// TIA Portal V17 export
// export: Created 2022-03-12T16:05:26.7716914Z, ExportSetting WithDefaults, DisplayName Totally Integrated Automation Portal, DisplayVersion V17, DisplayName TIA Portal Openness, DisplayVersion V17, DisplayName TIA Portal Version Control Interface, DisplayVersion V17, DisplayName STEP 7 Professional, DisplayVersion V17, DisplayName STEP 7 Safety, DisplayVersion V17, DisplayName WinCC Advanced / Unified PC, DisplayVersion V17
FUNCTION_BLOCK "EM00_CM01_MainOpStation"   // FB31651, LAD
TITLE = EM00_CM01_MainOpStation
{ S7_Optimized_Access := 'TRUE' }
AUTHOR : tech.team.motioncontrol@siemens.com
FAMILY : CPG
VERSION : 1.1
// Support: tech.team.motioncontrol@siemens.com
// stored: AutoNumber true, IsIECCheckEnabled false, IsRetainMemResEnabled false, MemoryReserve 100, SetENOAutomatically false, UDAEnableTagReadback false
   VAR
      instAlarm_EStop { ExternalAccessible := 'False'; ExternalVisible := 'False'; ExternalWritable := 'False'; S7_SetPoint := 'True'} : "CPG_Event";   // Alarm Event - EStop pressed (Event instance)
      instAlarm_HMI_StopPB { ExternalAccessible := 'False'; ExternalVisible := 'False'; ExternalWritable := 'False'; S7_SetPoint := 'True'} : "CPG_Event";   // Alarm Event - HMI Stop PB pressed (Event instance)
      instStatus_WaitingForStartCmd { ExternalAccessible := 'False'; ExternalVisible := 'False'; ExternalWritable := 'False'; S7_SetPoint := 'True'} : "CPG_Event";   // Status Event - waiting for start command (Event instance)
      instStatus_WaitingForResetCmd { ExternalAccessible := 'False'; ExternalVisible := 'False'; ExternalWritable := 'False'; S7_SetPoint := 'True'} : "CPG_Event";   // Status Event - waiting for reset command (Event instance)
      instAlarm_Hold_PB { ExternalAccessible := 'False'; ExternalVisible := 'False'; ExternalWritable := 'False'; S7_SetPoint := 'True'} : "CPG_Event";   // Alarm Event - HMI Held PB pressed (Event instance)
      instStatus_WaitingForUnHoldCmd { ExternalAccessible := 'False'; ExternalVisible := 'False'; ExternalWritable := 'False'; S7_SetPoint := 'True'} : "CPG_Event";   // Status Event - waiting for unhold command (Event instance)
      instTimer_StartingDelay_SC { ExternalAccessible := 'False'; ExternalVisible := 'False'; ExternalWritable := 'False'; S7_SetPoint := 'True'} : IEC_TIMER;   // IEC Timer - starting delay (demo only - used to slow state model transition)
      instTimer_CompletingDelay_SC { ExternalAccessible := 'False'; ExternalVisible := 'False'; ExternalWritable := 'False'; S7_SetPoint := 'True'} : IEC_TIMER;   // IEC Timer - completing delay (demo only - used to slow state model transition)
      instTimer_AbortingDelay_SC { ExternalAccessible := 'False'; ExternalVisible := 'False'; ExternalWritable := 'False'; S7_SetPoint := 'True'} : IEC_TIMER;   // IEC Timer - aborting delay (demo only - used to slow state model transition)
      instTimer_StoppingDelay_SC { ExternalAccessible := 'False'; ExternalVisible := 'False'; ExternalWritable := 'False'; S7_SetPoint := 'True'} : IEC_TIMER;   // IEC Timer - stopping delay (demo only - used to slow state model transition)
      instTimer_ResettingDelay_SC { ExternalAccessible := 'False'; ExternalVisible := 'False'; ExternalWritable := 'False'; S7_SetPoint := 'True'} : IEC_TIMER;   // IEC Timer - resetting delay (demo only - used to slow state model transition)
      instTimer_HoldingDelay_SC { ExternalAccessible := 'False'; ExternalVisible := 'False'; ExternalWritable := 'False'; S7_SetPoint := 'True'} : IEC_TIMER;   // IEC Timer - holding delay (demo only - used to slow state model transition)
      instTimer_UnHoldingDelay_SC { ExternalAccessible := 'False'; ExternalVisible := 'False'; ExternalWritable := 'False'; S7_SetPoint := 'True'} : IEC_TIMER;   // IEC Timer - un-holding delay (demo only - used to slow state model transition)
      instTimer_SuspendingDelay_SC { ExternalAccessible := 'False'; ExternalVisible := 'False'; ExternalWritable := 'False'; S7_SetPoint := 'True'} : IEC_TIMER;   // IEC Timer - suspending delay (demo only - used to slow state model transition)
      instTimer_UnSuspendingDelay_SC { ExternalAccessible := 'False'; ExternalVisible := 'False'; ExternalWritable := 'False'; S7_SetPoint := 'True'} : IEC_TIMER;   // IEC Timer - un-suspending delay (demo only - used to slow state model transition)
      instTimer_ClearingDelay_SC { ExternalAccessible := 'False'; ExternalVisible := 'False'; ExternalWritable := 'False'; S7_SetPoint := 'True'} : IEC_TIMER;   // IEC Timer - clearing delay (demo only - used to slow state model transition)
   END_VAR
BEGIN

REGION Network 1: *** Begin the Setpoint Management Information Section ***
END_REGION

REGION Network 2: *** Begin the Logic Section ***
END_REGION

REGION Network 3: *** Begin the Event Information Section ***
END_REGION

REGION Network 4: Alarm Event - EStop
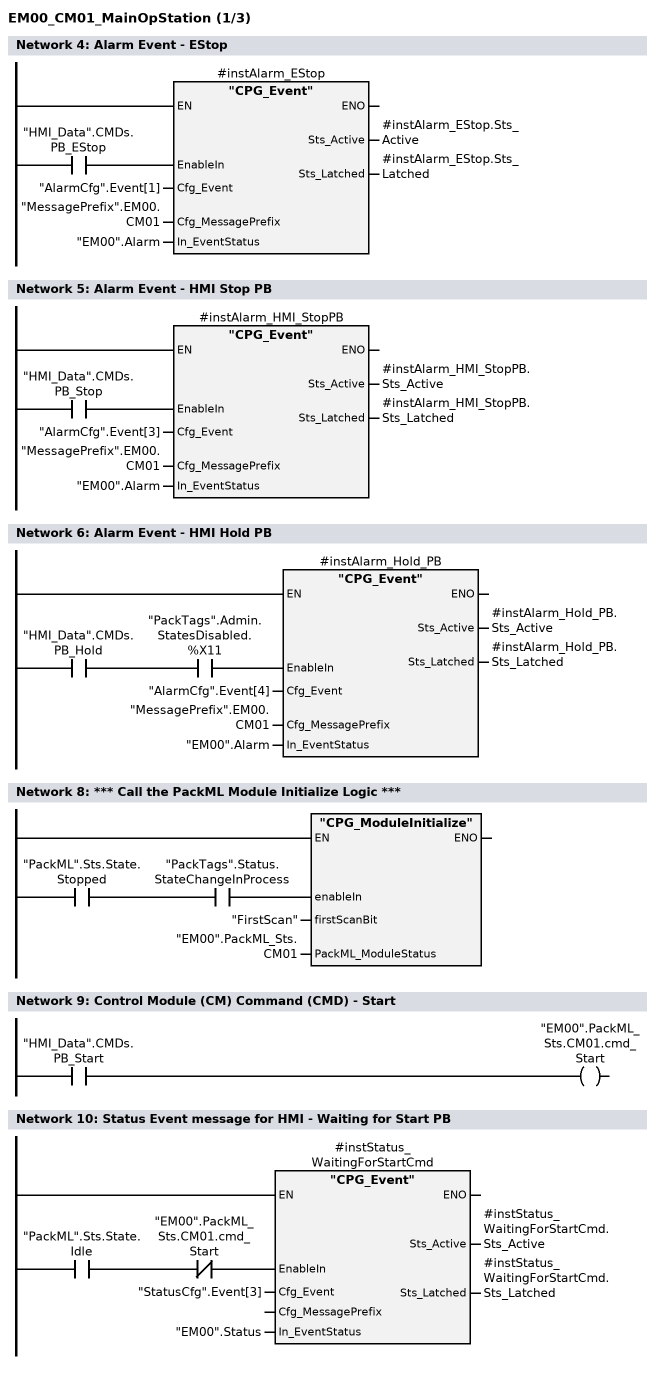
   RUNG wire#powerrail
      #instAlarm_EStop(EnableIn := wire#w1, Cfg_Event := "AlarmCfg".Event[1], Cfg_MessagePrefix := "MessagePrefix".EM00.CM01, In_EventStatus := "EM00".Alarm, Sts_Active => #instAlarm_EStop.Sts_Active, Sts_Latched => #instAlarm_EStop.Sts_Latched)
   END_RUNG
   RUNG wire#powerrail
      Contact( "HMI_Data".CMDs.PB_EStop )
   END_RUNG wire#w1
   // the same network as SCL:
   #instAlarm_EStop(EnableIn := "HMI_Data".CMDs.PB_EStop,   // "CPG_Event"
                    Cfg_Event := "AlarmCfg".Event[1],
                    Cfg_MessagePrefix := "MessagePrefix".EM00.CM01,
                    In_EventStatus := "EM00".Alarm,
                    Sts_Active => #instAlarm_EStop.Sts_Active,
                    Sts_Latched => #instAlarm_EStop.Sts_Latched);
END_REGION

REGION Network 5: Alarm Event - HMI Stop PB
   RUNG wire#powerrail
      #instAlarm_HMI_StopPB(EnableIn := wire#w1, Cfg_Event := "AlarmCfg".Event[3], Cfg_MessagePrefix := "MessagePrefix".EM00.CM01, In_EventStatus := "EM00".Alarm, Sts_Active => #instAlarm_HMI_StopPB.Sts_Active, Sts_Latched => #instAlarm_HMI_StopPB.Sts_Latched)
   END_RUNG
   RUNG wire#powerrail
      Contact( "HMI_Data".CMDs.PB_Stop )
   END_RUNG wire#w1
   // the same network as SCL:
   #instAlarm_HMI_StopPB(EnableIn := "HMI_Data".CMDs.PB_Stop,   // "CPG_Event"
                         Cfg_Event := "AlarmCfg".Event[3],
                         Cfg_MessagePrefix := "MessagePrefix".EM00.CM01,
                         In_EventStatus := "EM00".Alarm,
                         Sts_Active => #instAlarm_HMI_StopPB.Sts_Active,
                         Sts_Latched => #instAlarm_HMI_StopPB.Sts_Latched);
END_REGION

REGION Network 6: Alarm Event - HMI Hold PB
   RUNG wire#powerrail
      #instAlarm_Hold_PB(EnableIn := wire#w1, Cfg_Event := "AlarmCfg".Event[4], Cfg_MessagePrefix := "MessagePrefix".EM00.CM01, In_EventStatus := "EM00".Alarm, Sts_Active => #instAlarm_Hold_PB.Sts_Active, Sts_Latched => #instAlarm_Hold_PB.Sts_Latched)
   END_RUNG
   RUNG wire#powerrail
      Contact( "HMI_Data".CMDs.PB_Hold )
      Contact( "PackTags".Admin.StatesDisabled.%X11 )
   END_RUNG wire#w1
   // the same network as SCL:
   #instAlarm_Hold_PB(EnableIn := "HMI_Data".CMDs.PB_Hold AND "PackTags".Admin.StatesDisabled.%X11,   // "CPG_Event"
                      Cfg_Event := "AlarmCfg".Event[4],
                      Cfg_MessagePrefix := "MessagePrefix".EM00.CM01,
                      In_EventStatus := "EM00".Alarm,
                      Sts_Active => #instAlarm_Hold_PB.Sts_Active,
                      Sts_Latched => #instAlarm_Hold_PB.Sts_Latched);
END_REGION

REGION Network 7: *** Begin the State Model Status Feedback Section ***
END_REGION

REGION Network 8: *** Call the PackML Module Initialize Logic ***
   RUNG wire#powerrail
      "CPG_ModuleInitialize"(enableIn := wire#w1, firstScanBit := "FirstScan", PackML_ModuleStatus := "EM00".PackML_Sts.CM01)
   END_RUNG
   RUNG wire#powerrail
      Contact( "PackML".Sts.State.Stopped )
      Contact( "PackTags".Status.StateChangeInProcess )
   END_RUNG wire#w1
   // the same network as SCL:
   "CPG_ModuleInitialize"(enableIn := "PackML".Sts.State.Stopped AND "PackTags".Status.StateChangeInProcess,
                          firstScanBit := "FirstScan",
                          PackML_ModuleStatus := "EM00".PackML_Sts.CM01);
END_REGION

REGION Network 9: Control Module (CM) Command (CMD) - Start
   RUNG wire#powerrail
      Contact( "HMI_Data".CMDs.PB_Start )
      Coil( "EM00".PackML_Sts.CM01.cmd_Start )
   END_RUNG
   // the same network as SCL:
   "EM00".PackML_Sts.CM01.cmd_Start := "HMI_Data".CMDs.PB_Start;
END_REGION

REGION Network 10: Status Event message for HMI - Waiting for Start PB
   RUNG wire#powerrail
      #instStatus_WaitingForStartCmd(EnableIn := wire#w1, Cfg_Event := "StatusCfg".Event[3], Cfg_MessagePrefix :=, In_EventStatus := "EM00".Status, Sts_Active => #instStatus_WaitingForStartCmd.Sts_Active, Sts_Latched => #instStatus_WaitingForStartCmd.Sts_Latched)
   END_RUNG
   RUNG wire#powerrail
      Contact( "PackML".Sts.State.Idle )
      I_Contact( "EM00".PackML_Sts.CM01.cmd_Start )
   END_RUNG wire#w1
   // the same network as SCL:
   #instStatus_WaitingForStartCmd(EnableIn := "PackML".Sts.State.Idle AND NOT "EM00".PackML_Sts.CM01.cmd_Start,   // "CPG_Event"
                           Cfg_Event := "StatusCfg".Event[3],
                           In_EventStatus := "EM00".Status,
                           Sts_Active => #instStatus_WaitingForStartCmd.Sts_Active,
                           Sts_Latched => #instStatus_WaitingForStartCmd.Sts_Latched);
END_REGION

REGION Network 11: Control Module (CM) Command (CMD) - reset and clear commands
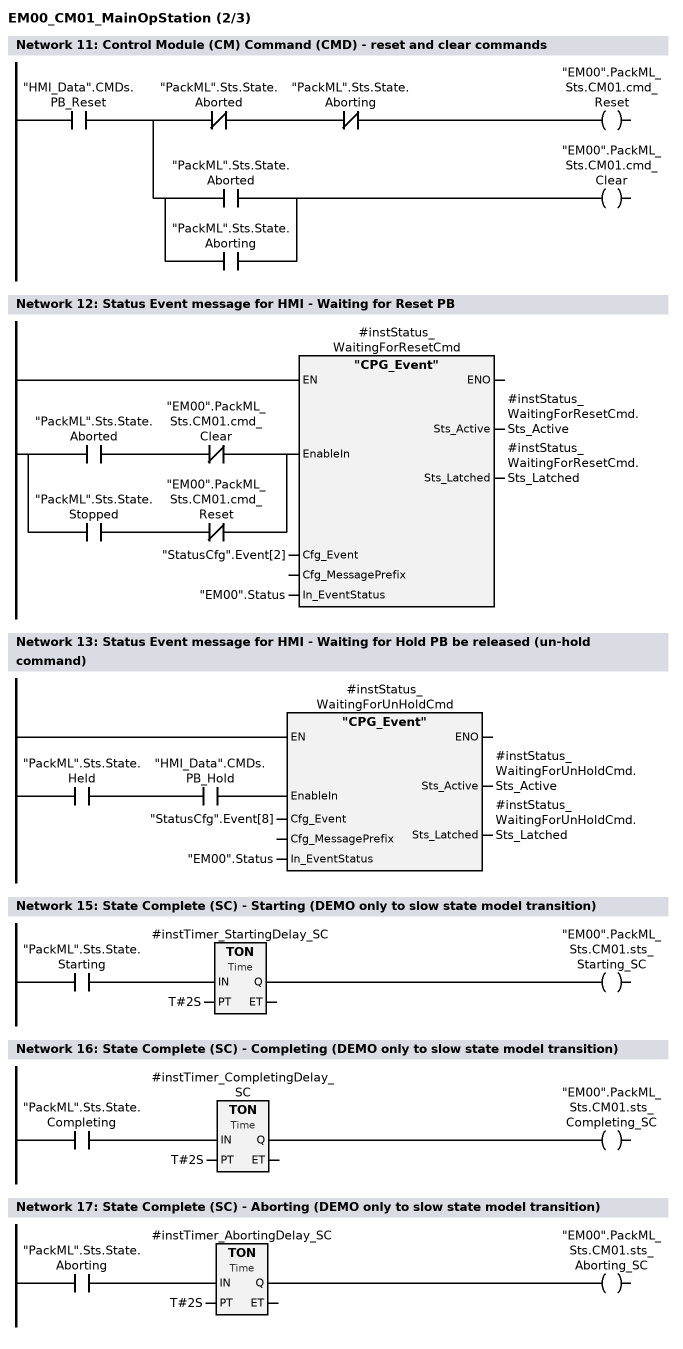
   RUNG wire#powerrail
      Contact( "HMI_Data".CMDs.PB_Reset )
      wire#w1
      I_Contact( "PackML".Sts.State.Aborted )
      I_Contact( "PackML".Sts.State.Aborting )
      Coil( "EM00".PackML_Sts.CM01.cmd_Reset )
   END_RUNG
   RUNG wire#w1
      Contact( "PackML".Sts.State.Aborted )
      wire#w2
      Coil( "EM00".PackML_Sts.CM01.cmd_Clear )
   END_RUNG
   RUNG wire#w1
      Contact( "PackML".Sts.State.Aborting )
   END_RUNG wire#w2
   // the same network as SCL:
   "EM00".PackML_Sts.CM01.cmd_Reset := "HMI_Data".CMDs.PB_Reset AND NOT "PackML".Sts.State.Aborted AND NOT "PackML".Sts.State.Aborting;
   "EM00".PackML_Sts.CM01.cmd_Clear := "HMI_Data".CMDs.PB_Reset AND ("PackML".Sts.State.Aborted OR "PackML".Sts.State.Aborting);
END_REGION

REGION Network 12: Status Event message for HMI - Waiting for Reset PB
   RUNG wire#powerrail
      #instStatus_WaitingForResetCmd(EnableIn := wire#w1, Cfg_Event := "StatusCfg".Event[2], Cfg_MessagePrefix :=, In_EventStatus := "EM00".Status, Sts_Active => #instStatus_WaitingForResetCmd.Sts_Active, Sts_Latched => #instStatus_WaitingForResetCmd.Sts_Latched)
   END_RUNG
   RUNG wire#powerrail
      Contact( "PackML".Sts.State.Aborted )
      I_Contact( "EM00".PackML_Sts.CM01.cmd_Clear )
   END_RUNG wire#w1
   RUNG wire#powerrail
      Contact( "PackML".Sts.State.Stopped )
      I_Contact( "EM00".PackML_Sts.CM01.cmd_Reset )
   END_RUNG wire#w1
   // the same network as SCL:
   #instStatus_WaitingForResetCmd(EnableIn := ("PackML".Sts.State.Aborted AND NOT "EM00".PackML_Sts.CM01.cmd_Clear) OR ("PackML".Sts.State.Stopped AND NOT "EM00".PackML_Sts.CM01.cmd_Reset),   // "CPG_Event"
                           Cfg_Event := "StatusCfg".Event[2],
                           In_EventStatus := "EM00".Status,
                           Sts_Active => #instStatus_WaitingForResetCmd.Sts_Active,
                           Sts_Latched => #instStatus_WaitingForResetCmd.Sts_Latched);
END_REGION

REGION Network 13: Status Event message for HMI - Waiting for Hold PB be released (un-hold command)
   RUNG wire#powerrail
      #instStatus_WaitingForUnHoldCmd(EnableIn := wire#w1, Cfg_Event := "StatusCfg".Event[8], Cfg_MessagePrefix :=, In_EventStatus := "EM00".Status, Sts_Active => #instStatus_WaitingForUnHoldCmd.Sts_Active, Sts_Latched => #instStatus_WaitingForUnHoldCmd.Sts_Latched)
   END_RUNG
   RUNG wire#powerrail
      Contact( "PackML".Sts.State.Held )
      Contact( "HMI_Data".CMDs.PB_Hold )
   END_RUNG wire#w1
   // the same network as SCL:
   #instStatus_WaitingForUnHoldCmd(EnableIn := "PackML".Sts.State.Held AND "HMI_Data".CMDs.PB_Hold,   // "CPG_Event"
                           Cfg_Event := "StatusCfg".Event[8],
                           In_EventStatus := "EM00".Status,
                           Sts_Active => #instStatus_WaitingForUnHoldCmd.Sts_Active,
                           Sts_Latched => #instStatus_WaitingForUnHoldCmd.Sts_Latched);
END_REGION

REGION Network 14: State Model delay timers used to slow state model transition - only used for demo purposes (remove for real projects)
END_REGION

REGION Network 15: State Complete (SC) - Starting (DEMO only to slow state model transition)
   RUNG wire#powerrail
      Contact( "PackML".Sts.State.Starting )
      { S7_Templates := "time_type := Time" } #instTimer_StartingDelay_SC.TON(pt := T#2S, et =>)
      Coil( "EM00".PackML_Sts.CM01.sts_Starting_SC )
   END_RUNG
   // the same network as SCL:
   #instTimer_StartingDelay_SC.TON(IN := "PackML".Sts.State.Starting, PT := T#2S);
   "EM00".PackML_Sts.CM01.sts_Starting_SC := #instTimer_StartingDelay_SC.Q;
END_REGION

REGION Network 16: State Complete (SC) - Completing (DEMO only to slow state model transition)
   RUNG wire#powerrail
      Contact( "PackML".Sts.State.Completing )
      { S7_Templates := "time_type := Time" } #instTimer_CompletingDelay_SC.TON(pt := T#2S, et =>)
      Coil( "EM00".PackML_Sts.CM01.sts_Completing_SC )
   END_RUNG
   // the same network as SCL:
   #instTimer_CompletingDelay_SC.TON(IN := "PackML".Sts.State.Completing, PT := T#2S);
   "EM00".PackML_Sts.CM01.sts_Completing_SC := #instTimer_CompletingDelay_SC.Q;
END_REGION

REGION Network 17: State Complete (SC) - Aborting (DEMO only to slow state model transition)
   RUNG wire#powerrail
      Contact( "PackML".Sts.State.Aborting )
      { S7_Templates := "time_type := Time" } #instTimer_AbortingDelay_SC.TON(pt := T#2S, et =>)
      Coil( "EM00".PackML_Sts.CM01.sts_Aborting_SC )
   END_RUNG
   // the same network as SCL:
   #instTimer_AbortingDelay_SC.TON(IN := "PackML".Sts.State.Aborting, PT := T#2S);
   "EM00".PackML_Sts.CM01.sts_Aborting_SC := #instTimer_AbortingDelay_SC.Q;
END_REGION

REGION Network 18: State Complete (SC) - Stopping (DEMO only to slow state model transition)
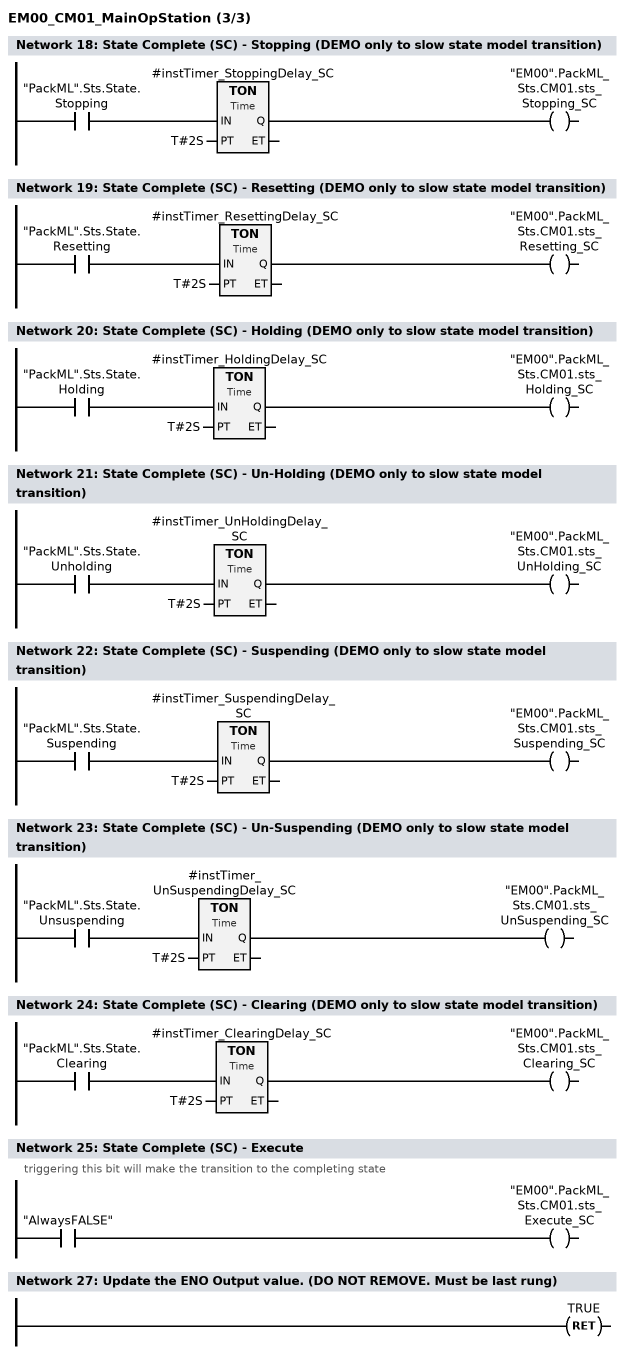
   RUNG wire#powerrail
      Contact( "PackML".Sts.State.Stopping )
      { S7_Templates := "time_type := Time" } #instTimer_StoppingDelay_SC.TON(pt := T#2S, et =>)
      Coil( "EM00".PackML_Sts.CM01.sts_Stopping_SC )
   END_RUNG
   // the same network as SCL:
   #instTimer_StoppingDelay_SC.TON(IN := "PackML".Sts.State.Stopping, PT := T#2S);
   "EM00".PackML_Sts.CM01.sts_Stopping_SC := #instTimer_StoppingDelay_SC.Q;
END_REGION

REGION Network 19: State Complete (SC) - Resetting (DEMO only to slow state model transition)
   RUNG wire#powerrail
      Contact( "PackML".Sts.State.Resetting )
      { S7_Templates := "time_type := Time" } #instTimer_ResettingDelay_SC.TON(pt := T#2S, et =>)
      Coil( "EM00".PackML_Sts.CM01.sts_Resetting_SC )
   END_RUNG
   // the same network as SCL:
   #instTimer_ResettingDelay_SC.TON(IN := "PackML".Sts.State.Resetting, PT := T#2S);
   "EM00".PackML_Sts.CM01.sts_Resetting_SC := #instTimer_ResettingDelay_SC.Q;
END_REGION

REGION Network 20: State Complete (SC) - Holding (DEMO only to slow state model transition)
   RUNG wire#powerrail
      Contact( "PackML".Sts.State.Holding )
      { S7_Templates := "time_type := Time" } #instTimer_HoldingDelay_SC.TON(pt := T#2S, et =>)
      Coil( "EM00".PackML_Sts.CM01.sts_Holding_SC )
   END_RUNG
   // the same network as SCL:
   #instTimer_HoldingDelay_SC.TON(IN := "PackML".Sts.State.Holding, PT := T#2S);
   "EM00".PackML_Sts.CM01.sts_Holding_SC := #instTimer_HoldingDelay_SC.Q;
END_REGION

REGION Network 21: State Complete (SC) - Un-Holding (DEMO only to slow state model transition)
   RUNG wire#powerrail
      Contact( "PackML".Sts.State.Unholding )
      { S7_Templates := "time_type := Time" } #instTimer_UnHoldingDelay_SC.TON(pt := T#2S, et =>)
      Coil( "EM00".PackML_Sts.CM01.sts_UnHolding_SC )
   END_RUNG
   // the same network as SCL:
   #instTimer_UnHoldingDelay_SC.TON(IN := "PackML".Sts.State.Unholding, PT := T#2S);
   "EM00".PackML_Sts.CM01.sts_UnHolding_SC := #instTimer_UnHoldingDelay_SC.Q;
END_REGION

REGION Network 22: State Complete (SC) - Suspending (DEMO only to slow state model transition)
   RUNG wire#powerrail
      Contact( "PackML".Sts.State.Suspending )
      { S7_Templates := "time_type := Time" } #instTimer_SuspendingDelay_SC.TON(pt := T#2S, et =>)
      Coil( "EM00".PackML_Sts.CM01.sts_Suspending_SC )
   END_RUNG
   // the same network as SCL:
   #instTimer_SuspendingDelay_SC.TON(IN := "PackML".Sts.State.Suspending, PT := T#2S);
   "EM00".PackML_Sts.CM01.sts_Suspending_SC := #instTimer_SuspendingDelay_SC.Q;
END_REGION

REGION Network 23: State Complete (SC) - Un-Suspending (DEMO only to slow state model transition)
   RUNG wire#powerrail
      Contact( "PackML".Sts.State.Unsuspending )
      { S7_Templates := "time_type := Time" } #instTimer_UnSuspendingDelay_SC.TON(pt := T#2S, et =>)
      Coil( "EM00".PackML_Sts.CM01.sts_UnSuspending_SC )
   END_RUNG
   // the same network as SCL:
   #instTimer_UnSuspendingDelay_SC.TON(IN := "PackML".Sts.State.Unsuspending, PT := T#2S);
   "EM00".PackML_Sts.CM01.sts_UnSuspending_SC := #instTimer_UnSuspendingDelay_SC.Q;
END_REGION

REGION Network 24: State Complete (SC) - Clearing (DEMO only to slow state model transition)
   RUNG wire#powerrail
      Contact( "PackML".Sts.State.Clearing )
      { S7_Templates := "time_type := Time" } #instTimer_ClearingDelay_SC.TON(pt := T#2S, et =>)
      Coil( "EM00".PackML_Sts.CM01.sts_Clearing_SC )
   END_RUNG
   // the same network as SCL:
   #instTimer_ClearingDelay_SC.TON(IN := "PackML".Sts.State.Clearing, PT := T#2S);
   "EM00".PackML_Sts.CM01.sts_Clearing_SC := #instTimer_ClearingDelay_SC.Q;
END_REGION

REGION Network 25: State Complete (SC) - Execute
   // triggering this bit will make the transition to the completing state
   RUNG wire#powerrail
      Contact( "AlwaysFALSE" )
      Coil( "EM00".PackML_Sts.CM01.sts_Execute_SC )
   END_RUNG
   // the same network as SCL:
   "EM00".PackML_Sts.CM01.sts_Execute_SC := "AlwaysFALSE";
END_REGION

REGION Network 27: Update the ENO Output value. (DO NOT REMOVE. Must be last rung)
   RUNG wire#powerrail
      ReturnCoil( TRUE )
   END_RUNG
   // the same network as SCL:
   ENO := TRUE;
   RETURN;
END_REGION
END_FUNCTION_BLOCK
